// TIA Portal V16 export
// export: Created 2021-08-10T09:04:59.634174Z, ExportSetting WithDefaults, WithReadOnly, DisplayName Totally Integrated Automation Portal, DisplayVersion V16, DisplayName TIA Portal Version Control Interface, DisplayVersion V16, DisplayName TIA Portal Openness, DisplayVersion V16, DisplayName TIA Portal Teamcenter Gateway, DisplayVersion V16, DisplayName SINAMICS Startdrive Advanced, DisplayVersion V16, DisplayName SINAMICS Startdrive G130, G150, S120, S150, SINAMICS MV, S210, DisplayVersion V16, DisplayName SINAMICS Startdrive G110M, G120, G120C, G120D, G120P, DisplayVersion V16, DisplayName STEP 7 Professional, DisplayVersion V16, DisplayName STEP 7 Safety, DisplayVersion V16, DisplayName WinCC Unified SCADA Engineering System, DisplayVersion V16
FUNCTION_BLOCK "Program Logic"   // FB5, FBD
{ S7_Optimized_Access := 'TRUE' }
VERSION : 0.1
// stored: AutoNumber true, CodeModifiedDate 2020-02-26T12:59:57.0334412Z, CompileDate 2021-07-03T08:38:44.9588418Z, CreationDate 2020-02-26T07:17:15.9384502Z, DownloadWithoutReinit false, HandleErrorsWithinBlock false, InterfaceModifiedDate 2020-02-26T11:20:20.4837101Z, IsConsistent true, IsIECCheckEnabled false, IsKnowHowProtected false, ISMultiInstanceCapable true, IsRetainMemResEnabled false, IsWriteProtected false, LibraryConformanceStatus Warning: The object contains access to global data blocks. Warning: The block contains direct access to inputs, outputs, bit memories, indirect access to the registry or indirect access to external memory areas that are unknown at the time of compilation., MemoryReserve 100, ModifiedDate 2020-02-26T12:59:57.0334412Z, ParameterModified 2020-02-26T07:17:15.9384502Z, PLCSimAdvancedSupport true, SetENOAutomatically false, StructureModified 2020-02-26T11:20:20.4837101Z, UDAEnableTagReadback false
   VAR
      StepSeq : "fbStepSequencer";
      CurrentStep { S7_SetPoint := 'True'} : Int;
      NextStep : Int;
      StepDone : Bool;
   END_VAR
   VAR_TEMP   // added for the SCL form of the ladder/FBD networks
      _w1 : Bool;
   END_VAR
BEGIN

REGION Network 1: 0 -- Idle
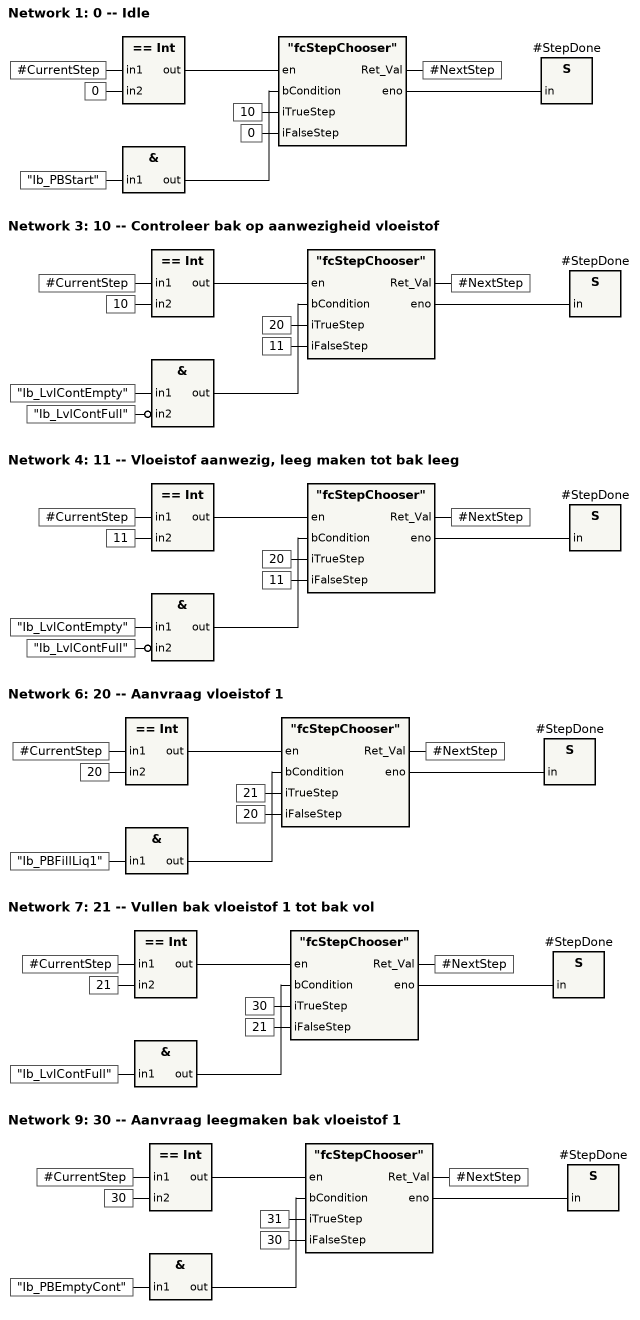
   #NextStep := "fcStepChooser"(EN := #CurrentStep = 0,
                           bCondition := "Ib_PBStart",
                           iTrueStep := 10,
                           iFalseStep := 0,
                           ENO => #_w1);
   IF #_w1 THEN #StepDone := TRUE; END_IF;
END_REGION

REGION Network 3: 10 -- Controleer bak op aanwezigheid vloeistof
   // vloeistof aanwezig 10->11
   // geen vloeistof aanwezig 10->20
   #NextStep := "fcStepChooser"(EN := #CurrentStep = 10,
                           bCondition := "Ib_LvlContEmpty" AND NOT "Ib_LvlContFull",
                           iTrueStep := 20,
                           iFalseStep := 11,
                           ENO => #_w1);
   IF #_w1 THEN #StepDone := TRUE; END_IF;
END_REGION

REGION Network 4: 11 -- Vloeistof aanwezig, leeg maken tot bak leeg
   #NextStep := "fcStepChooser"(EN := #CurrentStep = 11,
                           bCondition := "Ib_LvlContEmpty" AND NOT "Ib_LvlContFull",
                           iTrueStep := 20,
                           iFalseStep := 11,
                           ENO => #_w1);
   IF #_w1 THEN #StepDone := TRUE; END_IF;
END_REGION

REGION Network 6: 20 -- Aanvraag vloeistof 1
   #NextStep := "fcStepChooser"(EN := #CurrentStep = 20,
                           bCondition := "Ib_PBFillLiq1",
                           iTrueStep := 21,
                           iFalseStep := 20,
                           ENO => #_w1);
   IF #_w1 THEN #StepDone := TRUE; END_IF;
END_REGION

REGION Network 7: 21 -- Vullen bak vloeistof 1 tot bak vol
   #NextStep := "fcStepChooser"(EN := #CurrentStep = 21,
                           bCondition := "Ib_LvlContFull",
                           iTrueStep := 30,
                           iFalseStep := 21,
                           ENO => #_w1);
   IF #_w1 THEN #StepDone := TRUE; END_IF;
END_REGION

REGION Network 9: 30 -- Aanvraag leegmaken bak vloeistof 1
   #NextStep := "fcStepChooser"(EN := #CurrentStep = 30,
                           bCondition := "Ib_PBEmptyCont",
                           iTrueStep := 31,
                           iFalseStep := 30,
                           ENO => #_w1);
   IF #_w1 THEN #StepDone := TRUE; END_IF;
END_REGION

REGION Network 10: 31 -- Leeg maken bak vloeistof 1
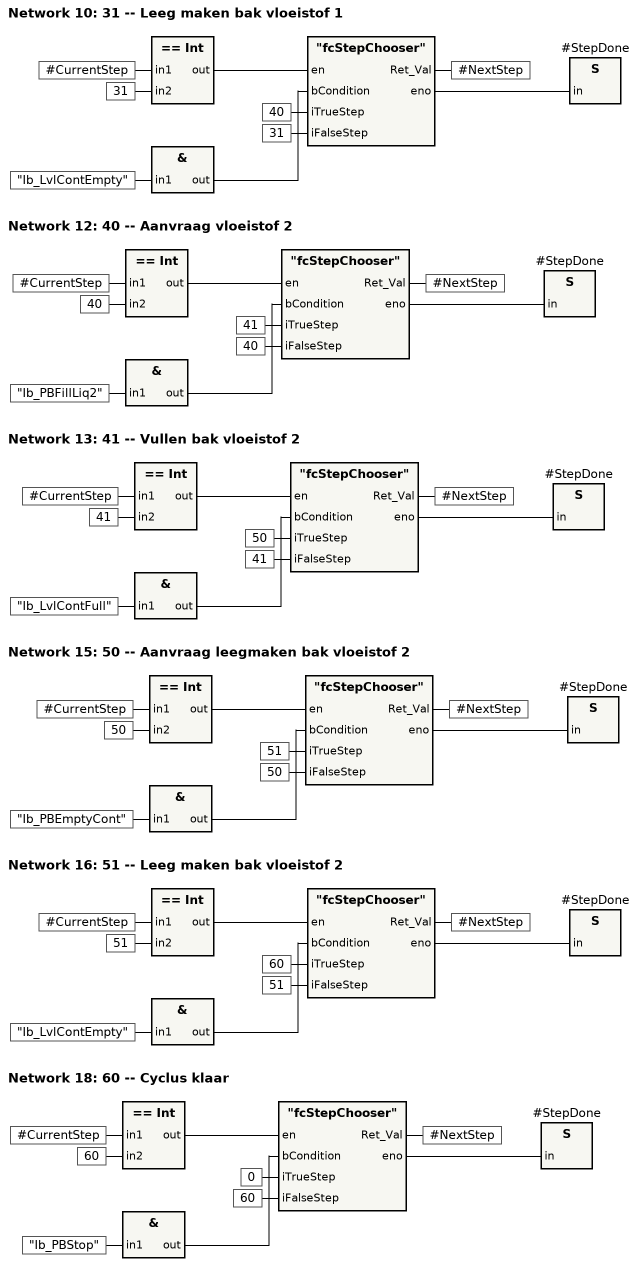
   #NextStep := "fcStepChooser"(EN := #CurrentStep = 31,
                           bCondition := "Ib_LvlContEmpty",
                           iTrueStep := 40,
                           iFalseStep := 31,
                           ENO => #_w1);
   IF #_w1 THEN #StepDone := TRUE; END_IF;
END_REGION

REGION Network 12: 40 -- Aanvraag vloeistof 2
   #NextStep := "fcStepChooser"(EN := #CurrentStep = 40,
                           bCondition := "Ib_PBFillLiq2",
                           iTrueStep := 41,
                           iFalseStep := 40,
                           ENO => #_w1);
   IF #_w1 THEN #StepDone := TRUE; END_IF;
END_REGION

REGION Network 13: 41 -- Vullen bak vloeistof 2
   #NextStep := "fcStepChooser"(EN := #CurrentStep = 41,
                           bCondition := "Ib_LvlContFull",
                           iTrueStep := 50,
                           iFalseStep := 41,
                           ENO => #_w1);
   IF #_w1 THEN #StepDone := TRUE; END_IF;
END_REGION

REGION Network 15: 50 -- Aanvraag leegmaken bak vloeistof 2
   #NextStep := "fcStepChooser"(EN := #CurrentStep = 50,
                           bCondition := "Ib_PBEmptyCont",
                           iTrueStep := 51,
                           iFalseStep := 50,
                           ENO => #_w1);
   IF #_w1 THEN #StepDone := TRUE; END_IF;
END_REGION

REGION Network 16: 51 -- Leeg maken bak vloeistof 2
   #NextStep := "fcStepChooser"(EN := #CurrentStep = 51,
                           bCondition := "Ib_LvlContEmpty",
                           iTrueStep := 60,
                           iFalseStep := 51,
                           ENO => #_w1);
   IF #_w1 THEN #StepDone := TRUE; END_IF;
END_REGION

REGION Network 18: 60 -- Cyclus klaar
   #NextStep := "fcStepChooser"(EN := #CurrentStep = 60,
                           bCondition := "Ib_PBStop",
                           iTrueStep := 0,
                           iFalseStep := 60,
                           ENO => #_w1);
   IF #_w1 THEN #StepDone := TRUE; END_IF;
END_REGION

REGION Network 20: Step Sequencer
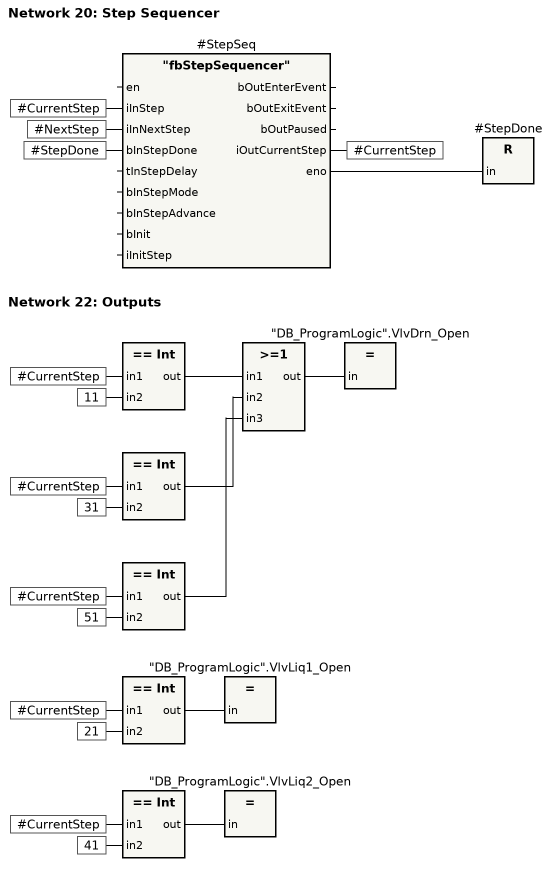
   #StepSeq(iInStep := #CurrentStep,   // "fbStepSequencer"
            iInNextStep := #NextStep,
            bInStepDone := #StepDone,
            iOutCurrentStep => #CurrentStep,
            ENO => #_w1);
   IF #_w1 THEN #StepDone := FALSE; END_IF;
END_REGION

REGION Network 22: Outputs
   "DB_ProgramLogic".VlvDrn_Open := (#CurrentStep = 11) OR (#CurrentStep = 31) OR (#CurrentStep = 51);
   "DB_ProgramLogic".VlvLiq1_Open := #CurrentStep = 21;
   "DB_ProgramLogic".VlvLiq2_Open := #CurrentStep = 41;
END_REGION
END_FUNCTION_BLOCK
